(* IEC 61131-3 sources: STM32_PLC/plc_examples, 3 files *)

(* ---- prog1_3btns.st ---- *)
PROGRAM PLC_PRG
  VAR_EXTERNAL
    pwm_out     : WORD;
    LCDText     : STRING; (* Global variable tied to %MD0 *)
    relay       : BOOL;
    btn_green   : BOOL;
    btn_red     : BOOL;
    btn_yellow  : BOOL;
  END_VAR

VAR
    (* Variables internes et détection de fronts *)
    btn_yellow_last : BOOL := FALSE;
    btn_green_last  : BOOL := FALSE;

    duty_cycle      : INT := 0;      (* Valeur de 0 à 100 *)
    prog_running    : BOOL := TRUE;  (* État du programme *)
END_VAR

(* Si le programme est running*)
IF prog_running THEN

    (* --- BOUTON VERT : Activation relais + Message --- *)

    IF btn_green THEN
        relay := TRUE;
        LCDtext := 'Green Btn OK';
    ELSE
        relay := FALSE;
        IF NOT btn_green AND btn_green_last THEN
           LCDtext := 'RELAY OFF';
        END_IF;
    END_IF;
    btn_green_last := btn_green;

    (* --- BOUTON JAUNE : Incrémentation PWM + Message --- *)
    (* Détection de 1 front montant (pression unique) *)
    IF btn_yellow AND NOT btn_yellow_last THEN

        (* Augmentation du duty cycle par pas de 10% avec plafond à 100% *)
        IF duty_cycle <= 100 THEN
            duty_cycle := duty_cycle + 10;
            IF duty_cycle > 100 THEN
                duty_cycle := 0;
            END_IF;
        END_IF;

        (* Application de la valeur sur la sortie PWM %QW0 *)
        pwm_out := INT_TO_WORD(DINT_TO_INT(INT_TO_DINT(duty_cycle) * 65535 / 100));

        (* dynamic Concatenation : "X% duty_cycle" *)
        LCDtext := CONCAT(INT_TO_STRING(duty_cycle), '% duty cycle');

    END_IF;
    btn_yellow_last := btn_yellow; (* Mémorisation état précédent *)

    (* --- BOUTON ROUGE : Arrêt du programme --- *)
    IF btn_red THEN
        relay := FALSE;
        pwm_out := 0;
        LCDtext := 'Program ended';
        prog_running := FALSE; (* Désactive le traitement principal *)
    END_IF;

END_IF;
END_PROGRAM

CONFIGURATION Config0

  RESOURCE Res0 ON PLC
    VAR_GLOBAL
      (* Entrées physiques *)
      btn_green  AT %IX0.0 : BOOL;
      btn_red    AT %IX0.1 : BOOL;
      btn_yellow AT %IX0.2 : BOOL;

      (* Sorties physiques *)
      relay      AT %QX0.2 : BOOL;
      pwm_out    AT %QW0   : WORD;

      (* Global variable bound to memory location %MD0 for hardware_layer.cpp *)
      LCDtext AT %MD0 : STRING := '3Btn+PWM1+DISP';
    END_VAR

    TASK TaskMain(INTERVAL := T#50ms, PRIORITY := 0);
    PROGRAM Inst0 WITH TaskMain : PLC_PRG;
  END_RESOURCE

END_CONFIGURATION

(* ---- testPWM1.st ---- *)
PROGRAM PWM_Tester
  VAR_EXTERNAL
    PWM1_Output : WORD;
    LCDText     : STRING; (* Global variable tied to %MD0 *)
  END_VAR

  VAR
    (* Timer to trigger state changes every 3 seconds *)
    StepTimer : TON;
    StepTimer_Q : BOOL;
    StepTimer_ET : TIME;

    (* Index tracking current duty cycle level (0 to 5) *)
    StepIndex : INT := 0;
  END_VAR

  (* -------------------------------------------------------------------
     1. TIMER LOGIC
     Runs continuously, pulsing StepTimer.Q high every 3.0 seconds
     ------------------------------------------------------------------- *)
  StepTimer(
    IN := NOT StepTimer.Q,
    PT := T#3s,
    Q => StepTimer_Q,
    ET => StepTimer_ET
  );

  (* -------------------------------------------------------------------
     2. STATE INCREMENT
     Advance to the next duty cycle level when timer completes
     ------------------------------------------------------------------- *)
  IF StepTimer.Q THEN
    StepIndex := StepIndex + 1;
    IF StepIndex > 5 THEN
      StepIndex := 0; (* Wrap back to 0% *)
    END_IF;
  END_IF;

  (* -------------------------------------------------------------------
     3. DUTY CYCLE LOOKUP, OUTPUT DRIVE & LCD UPDATE
     ------------------------------------------------------------------- *)
  CASE StepIndex OF
    0:
      PWM1_Output := UINT_TO_WORD(16#0000); (* 0% Duty *)
      LCDtext     := '0% Duty';
    1:
      PWM1_Output := UINT_TO_WORD(16#1999); (* 10% Duty *)
      LCDtext     := '10% Duty';
    2:
      PWM1_Output := UINT_TO_WORD(16#4CCD); (* 30% Duty *)
      LCDtext     := '30% Duty';
    3:
      PWM1_Output := UINT_TO_WORD(16#7FFF); (* 50% Duty *)
      LCDtext     := '50% Duty';
    4:
      PWM1_Output := UINT_TO_WORD(16#B332); (* 70% Duty *)
      LCDtext     := '70% Duty';
    5:
      PWM1_Output := UINT_TO_WORD(16#FFFF); (* 100% Duty *)
      LCDtext     := '100% Duty';
  ELSE
    StepIndex   := 0;
    PWM1_Output := UINT_TO_WORD(16#0000);
    LCDText     := 'Unknown Case';
  END_CASE;

END_PROGRAM

CONFIGURATION Config0

  RESOURCE Res0 ON PLC
    VAR_GLOBAL
      (* Hardware output mapped at global configuration scope *)
      PWM1_Output AT %QW0 : WORD;

      (* Global variable bound to memory location %MD0 for hardware_layer.cpp *)
      LCDtext AT %MD0 : STRING := 'Test PWM1';
    END_VAR

    TASK TaskMain(INTERVAL := T#50ms, PRIORITY := 0);
    PROGRAM Inst0 WITH TaskMain : PWM_Tester;
  END_RESOURCE

END_CONFIGURATION

(* ---- testRelays.st ---- *)
PROGRAM BlinkOUT10
  VAR_EXTERNAL
    REDLED : BOOL;
    ORANGELED : BOOL;
    RELAI0 : BOOL;
    RELAI1 : BOOL;
    RELAI2 : BOOL;
    IN1 : BOOL;
    LCDtext : STRING;
  END_VAR

  VAR
    IN1_prev : BOOL := FALSE;
    init_done : BOOL := FALSE;
    timer_red : TON;
    timer_orange : TON;
    led_state : BOOL := FALSE;
  END_VAR

  (* ------------------------------------------------------------- *)
  (* 1. INITIALIZATION ON FIRST SCAN                               *)
  (* ------------------------------------------------------------- *)
  IF NOT init_done THEN
    LCDtext := 'Loop Start';
    init_done := TRUE;
    IN1_prev := IN1;
  END_IF;

  (* ------------------------------------------------------------- *)
  (* 2. DYNAMIC LCD TEXT UPDATES (EDGE DETECTION)                 *)
  (* ------------------------------------------------------------- *)
  (* Detect Press (Rising Edge) *)
  IF IN1 AND NOT IN1_prev THEN
    LCDtext := 'Btn Pressed';
  END_IF;

  (* Detect Release (Falling Edge) *)
  IF NOT IN1 AND IN1_prev THEN
    LCDtext := 'Btn Released';
  END_IF;

  (* Store input state for next scan cycle *)
  IN1_prev := IN1;

  (* ------------------------------------------------------------- *)
  (* 3. LED & RELAY CONTROL LOGIC                                 *)
  (* ------------------------------------------------------------- *)
  IF IN1 THEN
    (* Flash RED LED and RELAI0 when button is pressed *)
    timer_red(IN := NOT timer_red.Q, PT := T#500ms);
    IF timer_red.Q THEN
      led_state := NOT led_state;
    END_IF;

    REDLED := led_state;
    RELAI0 := led_state;
    ORANGELED := FALSE;
    RELAI1 := FALSE;
  ELSE
    (* Flash ORANGE LED and RELAI1 when button is released *)
    timer_orange(IN := NOT timer_orange.Q, PT := T#1s);
    IF timer_orange.Q THEN
      led_state := NOT led_state;
    END_IF;

    ORANGELED := led_state;
    RELAI1 := led_state;
    REDLED := FALSE;
    RELAI0 := FALSE;
  END_IF;

END_PROGRAM

CONFIGURATION Config0
  RESOURCE Res0 ON PLC
    VAR_GLOBAL
      REDLED AT %QX1.0 : BOOL;
      ORANGELED AT %QX1.1 : BOOL;
      RELAI0 AT %QX0.0 : BOOL;
      RELAI1 AT %QX0.1 : BOOL;
      RELAI2 AT %QX0.2 : BOOL;
      IN1 AT %IX0.0 : BOOL;
      LCDtext AT %MD0 : STRING := 'OpenPLC V3\n';
    END_VAR
    TASK task0(INTERVAL := T#20ms, PRIORITY := 0);
    PROGRAM instance0 WITH task0 : BlinkOUT10;
  END_RESOURCE
END_CONFIGURATION
